FUNCTION_BLOCK PUBLIC RemainingTimeCalculator
VAR_INPUT
	elapsedSeconds : INT;
	elapsedMinutes : INT;
	givenDuration : INT; //Assume Duration in Minutes by default
END_VAR
VAR_OUTPUT
	leftOverSeconds : INT;
	leftOverMinutes : INT;
END_VAR
VAR
END_VAR

IF givenDuration <= elapsedMinutes THEN
	leftOverSeconds := 0;
	leftOverMinutes := 0;
ELSE
	leftOverMinutes := givenDuration - elapsedMinutes - 1;
	leftOverSeconds := 60 - elapsedSeconds;
END_IF

END_FUNCTION_BLOCK

(* stored: Version 1.1.0.1, ProductVersion 3.1.4024.3
   POU RemainingTimeCalculator: Id {dfca00c5-889e-49ff-92a2-6d9bf6d390bd}, SpecialFunc None *)
